(* PLC project Unnamed, Unknown Unnamed 1 *)
(* stored: creationDateTime 2021-05-11T15:41:27, modificationDateTime 2022-01-21T16:40:43 *)

PROGRAM SD_P
  VAR
    TIME_IN AT %MD0 : REAL;
    TIME_OUT AT %MD1 : REAL;
    SG1_Press AT %MD2 : REAL;
    SG2_Press AT %MD3 : REAL;
    SD_Valve AT %MD4 : REAL;
    SD_OnOff AT %MD5 : REAL := 0.0;
    MANIPIO_CONTROL AT %MD6 : REAL := 0.0;
    KPI AT %MD7 : REAL := 0.00005;
    Ti AT %MD8 : REAL := 20.0;
    SET_POINT AT %MD9 : REAL := 7692000.0;
    INIT AT %MD10 : REAL := 0.0;
  END_VAR
  VAR
    INTEGRAL0 : INTEGRAL;
  END_VAR
  VAR  (* added by the conversion: wires and edge detectors of the diagram *)
    _MUL7_OUT : REAL;
    _LIMIT18_OUT : ANY;
    _ADD14_OUT : ANY;
  END_VAR

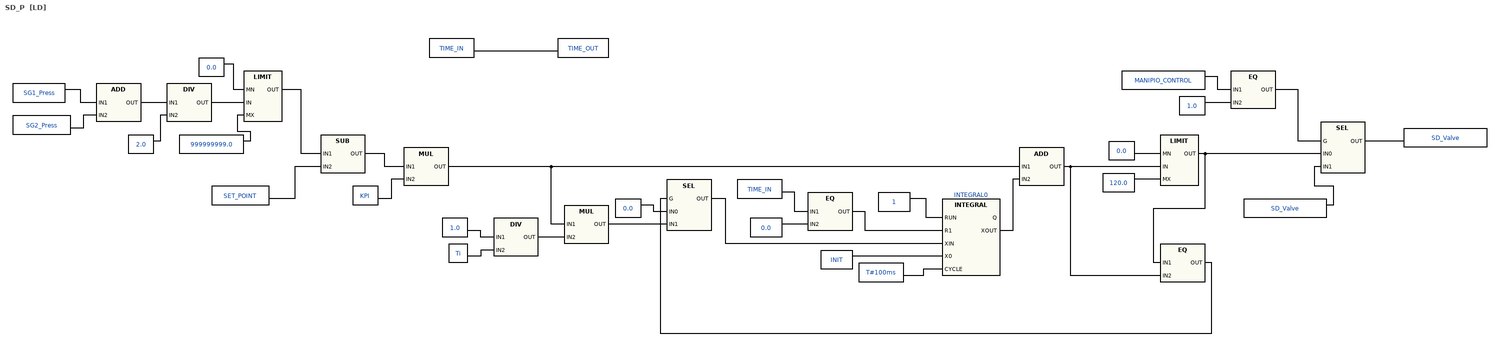
(* LD diagram, written out as Structured Text *)
TIME_OUT := TIME_IN;
_MUL7_OUT := (LIMIT(0.0, (SG1_Press + SG2_Press) / 2.0, 999999999.0) - SET_POINT) * KPI;
INTEGRAL0(RUN := 1, R1 := TIME_IN = 0.0, XIN := SEL(_LIMIT18_OUT = _ADD14_OUT, 0.0, _MUL7_OUT * (1.0 / Ti)), X0 := INIT, CYCLE := T#100ms);
_ADD14_OUT := _MUL7_OUT + INTEGRAL0.XOUT;
_LIMIT18_OUT := LIMIT(0.0, _ADD14_OUT, 120.0);
SD_Valve := SEL(MANIPIO_CONTROL = 1.0, _LIMIT18_OUT, SD_Valve);
END_PROGRAM

CONFIGURATION Config0
  RESOURCE Res0 ON PLC
    TASK task0(INTERVAL := T#100ms, PRIORITY := 0);
    PROGRAM instance0 WITH task0 : SD_P;
  END_RESOURCE
END_CONFIGURATION
